// TIA Portal V16 program export: 0 tag tables, 0 data types, 0 data blocks, 4 code blocks (in call order from the OBs), 0 instance data blocks

ORGANIZATION_BLOCK "Main"   // OB1, LAD, ProgramCycle
TITLE = "Main Program Sweep (Cycle)"
{ S7_Optimized_Access := 'TRUE' }
VERSION : 0.1
// stored: AutoNumber true, IsIECCheckEnabled false, SetENOAutomatically false
   VAR_INPUT
      Initial_Call : Bool;   // Initial call of this OB
      Remanence : Bool;   // =True, if remanent data are available
   END_VAR
BEGIN

REGION Network 1
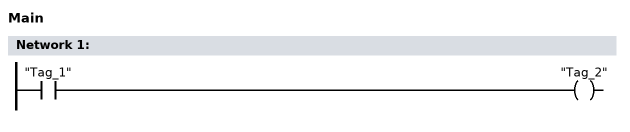
   RUNG wire#powerrail
      Contact( "Tag_1" )
      Coil( "Tag_2" )
   END_RUNG
   // the same network as SCL:
   "Tag_2" := "Tag_1";
END_REGION
END_ORGANIZATION_BLOCK

FUNCTION_BLOCK "FB1_TESTES"   // FB1, LAD
TITLE = FB para lógicas de testes durante start-up
{ S7_Optimized_Access := 'FALSE' }
AUTHOR : AUT_SIST
NAME : RGrn
VERSION : 0.1
// stored: AutoNumber false, IsIECCheckEnabled false, SetENOAutomatically false, UDAEnableTagReadback false
   VAR DB_SPECIFIC
      TESTE : Bool;
      bit_0_1 : Bool;
      bit_0_2 : Bool;
      bit_0_3 : Bool;
      bit_0_4 : Bool;
      bit_0_5 : Bool;
      bit_0_6 : Bool;
      bit_0_7 : Bool;
      bit_1_0 : Bool;
      bit_1_1 : Bool;
      bit_1_2 : Bool;
      bit_1_3 : Bool;
      bit_1_4 : Bool;
      bit_1_5 : Bool;
      bit_1_6 : Bool;
      bit_1_7 : Bool;
      eBosch_FO1_InCy : Bool;
      eBosch_FO1_CyCmp : Bool;
      eBosch_Ch0_1_OK : Bool;
      eBosch_Ch0_2_OK : Bool;
      eBosch_Ch0_3_OK : Bool;
      eBosch_Ch1_1_OK : Bool;
      eBosch_Ch1_2_OK : Bool;
      eBosch_Ch1_3_OK : Bool;
      eBosch_FO2_InCy : Bool;
      eBosch_FO2_CyCmp : Bool;
      eBosch_Ch2_1_OK : Bool;
      eBosch_Ch2_2_OK : Bool;
      eBosch_Ch2_3_OK : Bool;
      eBosch_Ch2_4_OK : Bool;
      bit_3_6 : Bool;
      bit_3_7 : Bool;
      bit_4_0 : Bool;
      bit_4_1 : Bool;
      bit_4_2 : Bool;
      bit_4_3 : Bool;
      bit_4_4 : Bool;
      bit_4_5 : Bool;
      bit_4_6 : Bool;
      bit_4_7 : Bool;
      FP_0 : Bool;
      FP_1 : Bool;
      FP_2 : Bool;
      FP_3 : Bool;
      FP_4 : Bool;
      FP_5 : Bool;
      FP_6 : Bool;
      FP_7 : Bool;
   END_VAR
   VAR_TEMP
      RET_VAL_FC455 : Word;
      Aux_Soma_rodas : Real;
      Med_Rot_rodas : Real;
      Med_parcial_rel_trm : Real;
      Retval_SFC20 : Int;   // Auxiliar armazenamento de mensagens do SFC20
      zero : DWord;
   END_VAR
BEGIN
END_FUNCTION_BLOCK

FUNCTION "FC180_STATUS" : Void   // FC180, LAD
TITLE = Status
{ S7_Optimized_Access := 'TRUE' }
VERSION : 0.1
// stored: AutoNumber false, IsIECCheckEnabled false, SetENOAutomatically false, UDAEnableTagReadback false
   VAR_TEMP
      DB180 : DB_ANY;
   END_VAR
BEGIN

REGION Network 1: DB_ANY CARREGA DB DE REFERENCIA NA VARIAVEL DE INDEXAÇÃO
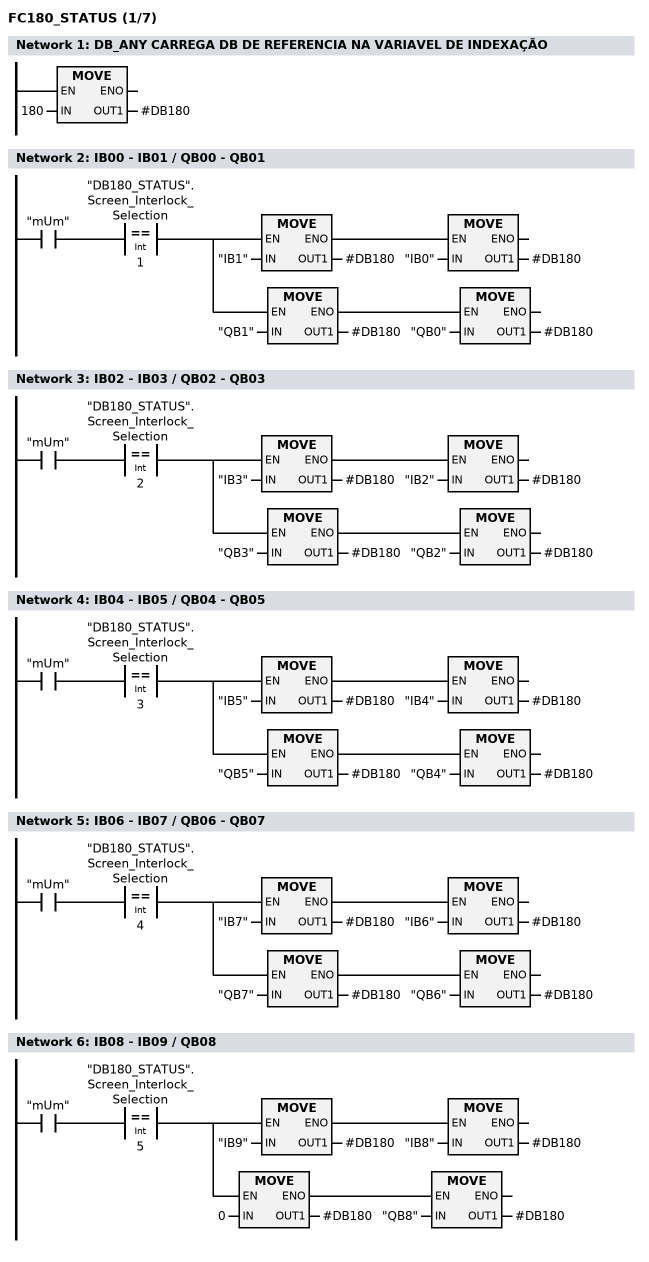
   RUNG wire#powerrail
      Move(in := 180, out1 => #DB180)
   END_RUNG
   // the same network as SCL:
   #DB180 := 180;
END_REGION

REGION Network 2: IB00 - IB01 / QB00 - QB01
   RUNG wire#powerrail
      Contact( "mUm" )
      { S7_Templates := "SrcType := Int" } EQ_Contact(in1 := "DB180_STATUS".Screen_Interlock_Selection, in2 := 1)
      wire#w1
      Move(in := "IB1", out1 => #DB180)
      Move(in := "IB0", out1 => #DB180)
   END_RUNG
   RUNG wire#w1
      Move(in := "QB1", out1 => #DB180)
      Move(in := "QB0", out1 => #DB180)
   END_RUNG
   // the same network as SCL:
   IF "mUm" AND ("DB180_STATUS".Screen_Interlock_Selection = 1) THEN
       #DB180 := "IB1";
       #DB180 := "IB0";
       #DB180 := "QB1";
       #DB180 := "QB0";
   END_IF;
END_REGION

REGION Network 3: IB02 - IB03 / QB02 - QB03
   RUNG wire#powerrail
      Contact( "mUm" )
      { S7_Templates := "SrcType := Int" } EQ_Contact(in1 := "DB180_STATUS".Screen_Interlock_Selection, in2 := 2)
      wire#w1
      Move(in := "IB3", out1 => #DB180)
      Move(in := "IB2", out1 => #DB180)
   END_RUNG
   RUNG wire#w1
      Move(in := "QB3", out1 => #DB180)
      Move(in := "QB2", out1 => #DB180)
   END_RUNG
   // the same network as SCL:
   IF "mUm" AND ("DB180_STATUS".Screen_Interlock_Selection = 2) THEN
       #DB180 := "IB3";
       #DB180 := "IB2";
       #DB180 := "QB3";
       #DB180 := "QB2";
   END_IF;
END_REGION

REGION Network 4: IB04 - IB05 / QB04 - QB05
   RUNG wire#powerrail
      Contact( "mUm" )
      { S7_Templates := "SrcType := Int" } EQ_Contact(in1 := "DB180_STATUS".Screen_Interlock_Selection, in2 := 3)
      wire#w1
      Move(in := "IB5", out1 => #DB180)
      Move(in := "IB4", out1 => #DB180)
   END_RUNG
   RUNG wire#w1
      Move(in := "QB5", out1 => #DB180)
      Move(in := "QB4", out1 => #DB180)
   END_RUNG
   // the same network as SCL:
   IF "mUm" AND ("DB180_STATUS".Screen_Interlock_Selection = 3) THEN
       #DB180 := "IB5";
       #DB180 := "IB4";
       #DB180 := "QB5";
       #DB180 := "QB4";
   END_IF;
END_REGION

REGION Network 5: IB06 - IB07 / QB06 - QB07
   RUNG wire#powerrail
      Contact( "mUm" )
      { S7_Templates := "SrcType := Int" } EQ_Contact(in1 := "DB180_STATUS".Screen_Interlock_Selection, in2 := 4)
      wire#w1
      Move(in := "IB7", out1 => #DB180)
      Move(in := "IB6", out1 => #DB180)
   END_RUNG
   RUNG wire#w1
      Move(in := "QB7", out1 => #DB180)
      Move(in := "QB6", out1 => #DB180)
   END_RUNG
   // the same network as SCL:
   IF "mUm" AND ("DB180_STATUS".Screen_Interlock_Selection = 4) THEN
       #DB180 := "IB7";
       #DB180 := "IB6";
       #DB180 := "QB7";
       #DB180 := "QB6";
   END_IF;
END_REGION

REGION Network 6: IB08 - IB09 / QB08
   RUNG wire#powerrail
      Contact( "mUm" )
      { S7_Templates := "SrcType := Int" } EQ_Contact(in1 := "DB180_STATUS".Screen_Interlock_Selection, in2 := 5)
      wire#w1
      Move(in := "IB9", out1 => #DB180)
      Move(in := "IB8", out1 => #DB180)
   END_RUNG
   RUNG wire#w1
      Move(in := 0, out1 => #DB180)
      Move(in := "QB8", out1 => #DB180)
   END_RUNG
   // the same network as SCL:
   IF "mUm" AND ("DB180_STATUS".Screen_Interlock_Selection = 5) THEN
       #DB180 := "IB9";
       #DB180 := "IB8";
       #DB180 := 0;
       #DB180 := "QB8";
   END_IF;
END_REGION

REGION Network 7: IB21 - IB23 / QB20 - QB22
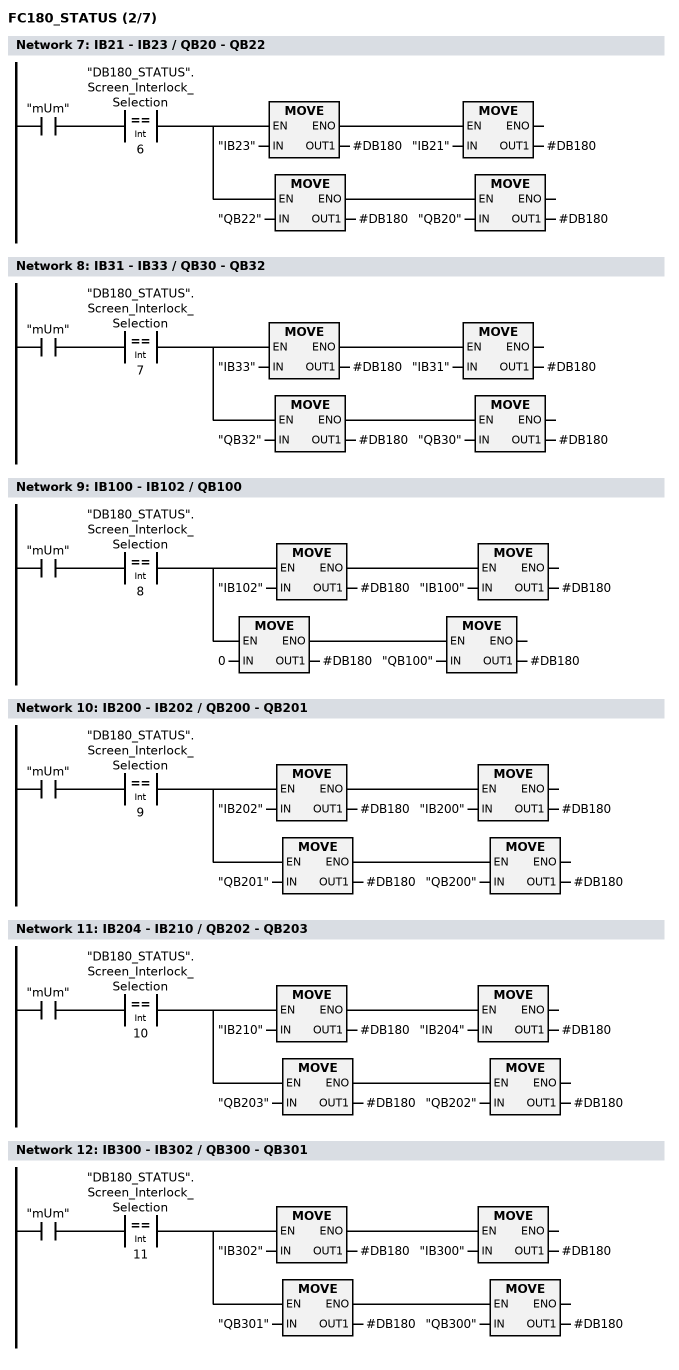
   RUNG wire#powerrail
      Contact( "mUm" )
      { S7_Templates := "SrcType := Int" } EQ_Contact(in1 := "DB180_STATUS".Screen_Interlock_Selection, in2 := 6)
      wire#w1
      Move(in := "IB23", out1 => #DB180)
      Move(in := "IB21", out1 => #DB180)
   END_RUNG
   RUNG wire#w1
      Move(in := "QB22", out1 => #DB180)
      Move(in := "QB20", out1 => #DB180)
   END_RUNG
   // the same network as SCL:
   IF "mUm" AND ("DB180_STATUS".Screen_Interlock_Selection = 6) THEN
       #DB180 := "IB23";
       #DB180 := "IB21";
       #DB180 := "QB22";
       #DB180 := "QB20";
   END_IF;
END_REGION

REGION Network 8: IB31 - IB33 / QB30 - QB32
   RUNG wire#powerrail
      Contact( "mUm" )
      { S7_Templates := "SrcType := Int" } EQ_Contact(in1 := "DB180_STATUS".Screen_Interlock_Selection, in2 := 7)
      wire#w1
      Move(in := "IB33", out1 => #DB180)
      Move(in := "IB31", out1 => #DB180)
   END_RUNG
   RUNG wire#w1
      Move(in := "QB32", out1 => #DB180)
      Move(in := "QB30", out1 => #DB180)
   END_RUNG
   // the same network as SCL:
   IF "mUm" AND ("DB180_STATUS".Screen_Interlock_Selection = 7) THEN
       #DB180 := "IB33";
       #DB180 := "IB31";
       #DB180 := "QB32";
       #DB180 := "QB30";
   END_IF;
END_REGION

REGION Network 9: IB100 - IB102 / QB100
   RUNG wire#powerrail
      Contact( "mUm" )
      { S7_Templates := "SrcType := Int" } EQ_Contact(in1 := "DB180_STATUS".Screen_Interlock_Selection, in2 := 8)
      wire#w1
      Move(in := "IB102", out1 => #DB180)
      Move(in := "IB100", out1 => #DB180)
   END_RUNG
   RUNG wire#w1
      Move(in := 0, out1 => #DB180)
      Move(in := "QB100", out1 => #DB180)
   END_RUNG
   // the same network as SCL:
   IF "mUm" AND ("DB180_STATUS".Screen_Interlock_Selection = 8) THEN
       #DB180 := "IB102";
       #DB180 := "IB100";
       #DB180 := 0;
       #DB180 := "QB100";
   END_IF;
END_REGION

REGION Network 10: IB200 - IB202 / QB200 - QB201
   RUNG wire#powerrail
      Contact( "mUm" )
      { S7_Templates := "SrcType := Int" } EQ_Contact(in1 := "DB180_STATUS".Screen_Interlock_Selection, in2 := 9)
      wire#w1
      Move(in := "IB202", out1 => #DB180)
      Move(in := "IB200", out1 => #DB180)
   END_RUNG
   RUNG wire#w1
      Move(in := "QB201", out1 => #DB180)
      Move(in := "QB200", out1 => #DB180)
   END_RUNG
   // the same network as SCL:
   IF "mUm" AND ("DB180_STATUS".Screen_Interlock_Selection = 9) THEN
       #DB180 := "IB202";
       #DB180 := "IB200";
       #DB180 := "QB201";
       #DB180 := "QB200";
   END_IF;
END_REGION

REGION Network 11: IB204 - IB210 / QB202 - QB203
   RUNG wire#powerrail
      Contact( "mUm" )
      { S7_Templates := "SrcType := Int" } EQ_Contact(in1 := "DB180_STATUS".Screen_Interlock_Selection, in2 := 10)
      wire#w1
      Move(in := "IB210", out1 => #DB180)
      Move(in := "IB204", out1 => #DB180)
   END_RUNG
   RUNG wire#w1
      Move(in := "QB203", out1 => #DB180)
      Move(in := "QB202", out1 => #DB180)
   END_RUNG
   // the same network as SCL:
   IF "mUm" AND ("DB180_STATUS".Screen_Interlock_Selection = 10) THEN
       #DB180 := "IB210";
       #DB180 := "IB204";
       #DB180 := "QB203";
       #DB180 := "QB202";
   END_IF;
END_REGION

REGION Network 12: IB300 - IB302 / QB300 - QB301
   RUNG wire#powerrail
      Contact( "mUm" )
      { S7_Templates := "SrcType := Int" } EQ_Contact(in1 := "DB180_STATUS".Screen_Interlock_Selection, in2 := 11)
      wire#w1
      Move(in := "IB302", out1 => #DB180)
      Move(in := "IB300", out1 => #DB180)
   END_RUNG
   RUNG wire#w1
      Move(in := "QB301", out1 => #DB180)
      Move(in := "QB300", out1 => #DB180)
   END_RUNG
   // the same network as SCL:
   IF "mUm" AND ("DB180_STATUS".Screen_Interlock_Selection = 11) THEN
       #DB180 := "IB302";
       #DB180 := "IB300";
       #DB180 := "QB301";
       #DB180 := "QB300";
   END_IF;
END_REGION

REGION Network 13: IB304 - IB306 / QB302 - QB303
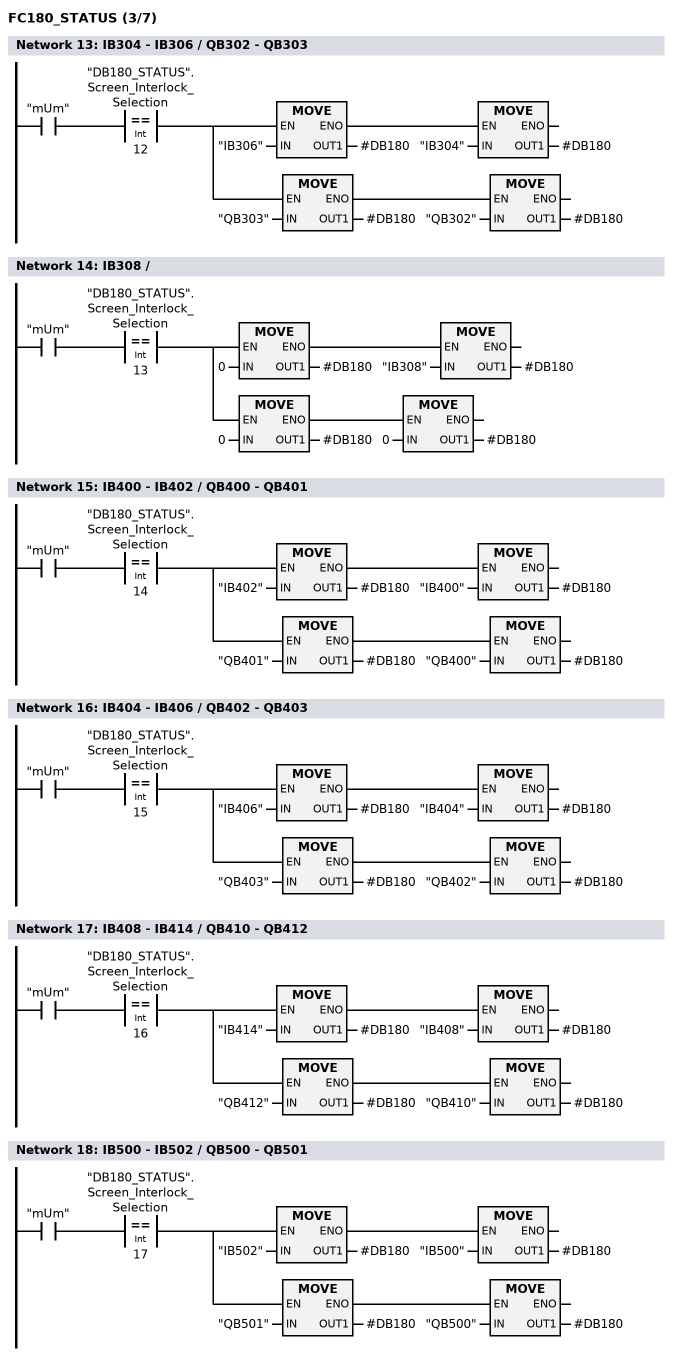
   RUNG wire#powerrail
      Contact( "mUm" )
      { S7_Templates := "SrcType := Int" } EQ_Contact(in1 := "DB180_STATUS".Screen_Interlock_Selection, in2 := 12)
      wire#w1
      Move(in := "IB306", out1 => #DB180)
      Move(in := "IB304", out1 => #DB180)
   END_RUNG
   RUNG wire#w1
      Move(in := "QB303", out1 => #DB180)
      Move(in := "QB302", out1 => #DB180)
   END_RUNG
   // the same network as SCL:
   IF "mUm" AND ("DB180_STATUS".Screen_Interlock_Selection = 12) THEN
       #DB180 := "IB306";
       #DB180 := "IB304";
       #DB180 := "QB303";
       #DB180 := "QB302";
   END_IF;
END_REGION

REGION Network 14: IB308 /
   RUNG wire#powerrail
      Contact( "mUm" )
      { S7_Templates := "SrcType := Int" } EQ_Contact(in1 := "DB180_STATUS".Screen_Interlock_Selection, in2 := 13)
      wire#w1
      Move(in := 0, out1 => #DB180)
      Move(in := "IB308", out1 => #DB180)
   END_RUNG
   RUNG wire#w1
      Move(in := 0, out1 => #DB180)
      Move(in := 0, out1 => #DB180)
   END_RUNG
   // the same network as SCL:
   IF "mUm" AND ("DB180_STATUS".Screen_Interlock_Selection = 13) THEN
       #DB180 := 0;
       #DB180 := "IB308";
       #DB180 := 0;
       #DB180 := 0;
   END_IF;
END_REGION

REGION Network 15: IB400 - IB402 / QB400 - QB401
   RUNG wire#powerrail
      Contact( "mUm" )
      { S7_Templates := "SrcType := Int" } EQ_Contact(in1 := "DB180_STATUS".Screen_Interlock_Selection, in2 := 14)
      wire#w1
      Move(in := "IB402", out1 => #DB180)
      Move(in := "IB400", out1 => #DB180)
   END_RUNG
   RUNG wire#w1
      Move(in := "QB401", out1 => #DB180)
      Move(in := "QB400", out1 => #DB180)
   END_RUNG
   // the same network as SCL:
   IF "mUm" AND ("DB180_STATUS".Screen_Interlock_Selection = 14) THEN
       #DB180 := "IB402";
       #DB180 := "IB400";
       #DB180 := "QB401";
       #DB180 := "QB400";
   END_IF;
END_REGION

REGION Network 16: IB404 - IB406 / QB402 - QB403
   RUNG wire#powerrail
      Contact( "mUm" )
      { S7_Templates := "SrcType := Int" } EQ_Contact(in1 := "DB180_STATUS".Screen_Interlock_Selection, in2 := 15)
      wire#w1
      Move(in := "IB406", out1 => #DB180)
      Move(in := "IB404", out1 => #DB180)
   END_RUNG
   RUNG wire#w1
      Move(in := "QB403", out1 => #DB180)
      Move(in := "QB402", out1 => #DB180)
   END_RUNG
   // the same network as SCL:
   IF "mUm" AND ("DB180_STATUS".Screen_Interlock_Selection = 15) THEN
       #DB180 := "IB406";
       #DB180 := "IB404";
       #DB180 := "QB403";
       #DB180 := "QB402";
   END_IF;
END_REGION

REGION Network 17: IB408 - IB414 / QB410 - QB412
   RUNG wire#powerrail
      Contact( "mUm" )
      { S7_Templates := "SrcType := Int" } EQ_Contact(in1 := "DB180_STATUS".Screen_Interlock_Selection, in2 := 16)
      wire#w1
      Move(in := "IB414", out1 => #DB180)
      Move(in := "IB408", out1 => #DB180)
   END_RUNG
   RUNG wire#w1
      Move(in := "QB412", out1 => #DB180)
      Move(in := "QB410", out1 => #DB180)
   END_RUNG
   // the same network as SCL:
   IF "mUm" AND ("DB180_STATUS".Screen_Interlock_Selection = 16) THEN
       #DB180 := "IB414";
       #DB180 := "IB408";
       #DB180 := "QB412";
       #DB180 := "QB410";
   END_IF;
END_REGION

REGION Network 18: IB500 - IB502 / QB500 - QB501
   RUNG wire#powerrail
      Contact( "mUm" )
      { S7_Templates := "SrcType := Int" } EQ_Contact(in1 := "DB180_STATUS".Screen_Interlock_Selection, in2 := 17)
      wire#w1
      Move(in := "IB502", out1 => #DB180)
      Move(in := "IB500", out1 => #DB180)
   END_RUNG
   RUNG wire#w1
      Move(in := "QB501", out1 => #DB180)
      Move(in := "QB500", out1 => #DB180)
   END_RUNG
   // the same network as SCL:
   IF "mUm" AND ("DB180_STATUS".Screen_Interlock_Selection = 17) THEN
       #DB180 := "IB502";
       #DB180 := "IB500";
       #DB180 := "QB501";
       #DB180 := "QB500";
   END_IF;
END_REGION

REGION Network 19: IB504 - IB506 / QB502 - QB503
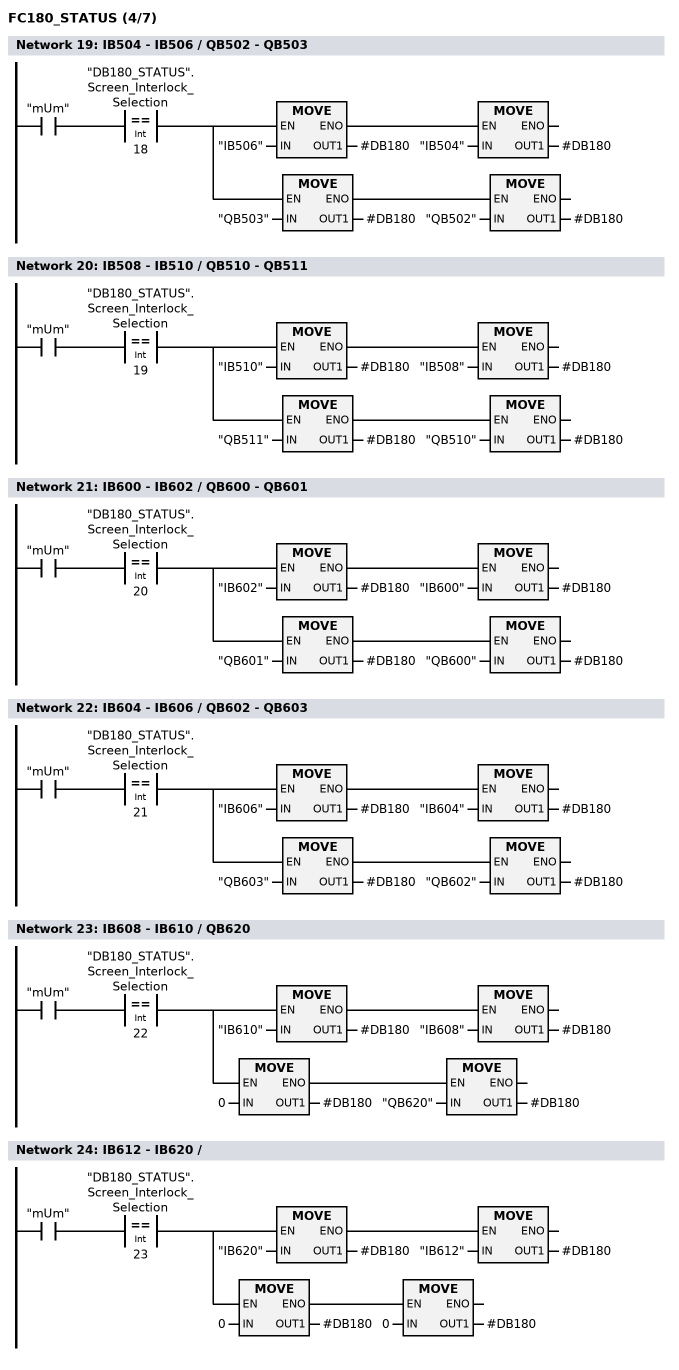
   RUNG wire#powerrail
      Contact( "mUm" )
      { S7_Templates := "SrcType := Int" } EQ_Contact(in1 := "DB180_STATUS".Screen_Interlock_Selection, in2 := 18)
      wire#w1
      Move(in := "IB506", out1 => #DB180)
      Move(in := "IB504", out1 => #DB180)
   END_RUNG
   RUNG wire#w1
      Move(in := "QB503", out1 => #DB180)
      Move(in := "QB502", out1 => #DB180)
   END_RUNG
   // the same network as SCL:
   IF "mUm" AND ("DB180_STATUS".Screen_Interlock_Selection = 18) THEN
       #DB180 := "IB506";
       #DB180 := "IB504";
       #DB180 := "QB503";
       #DB180 := "QB502";
   END_IF;
END_REGION

REGION Network 20: IB508 - IB510 / QB510 - QB511
   RUNG wire#powerrail
      Contact( "mUm" )
      { S7_Templates := "SrcType := Int" } EQ_Contact(in1 := "DB180_STATUS".Screen_Interlock_Selection, in2 := 19)
      wire#w1
      Move(in := "IB510", out1 => #DB180)
      Move(in := "IB508", out1 => #DB180)
   END_RUNG
   RUNG wire#w1
      Move(in := "QB511", out1 => #DB180)
      Move(in := "QB510", out1 => #DB180)
   END_RUNG
   // the same network as SCL:
   IF "mUm" AND ("DB180_STATUS".Screen_Interlock_Selection = 19) THEN
       #DB180 := "IB510";
       #DB180 := "IB508";
       #DB180 := "QB511";
       #DB180 := "QB510";
   END_IF;
END_REGION

REGION Network 21: IB600 - IB602 / QB600 - QB601
   RUNG wire#powerrail
      Contact( "mUm" )
      { S7_Templates := "SrcType := Int" } EQ_Contact(in1 := "DB180_STATUS".Screen_Interlock_Selection, in2 := 20)
      wire#w1
      Move(in := "IB602", out1 => #DB180)
      Move(in := "IB600", out1 => #DB180)
   END_RUNG
   RUNG wire#w1
      Move(in := "QB601", out1 => #DB180)
      Move(in := "QB600", out1 => #DB180)
   END_RUNG
   // the same network as SCL:
   IF "mUm" AND ("DB180_STATUS".Screen_Interlock_Selection = 20) THEN
       #DB180 := "IB602";
       #DB180 := "IB600";
       #DB180 := "QB601";
       #DB180 := "QB600";
   END_IF;
END_REGION

REGION Network 22: IB604 - IB606 / QB602 - QB603
   RUNG wire#powerrail
      Contact( "mUm" )
      { S7_Templates := "SrcType := Int" } EQ_Contact(in1 := "DB180_STATUS".Screen_Interlock_Selection, in2 := 21)
      wire#w1
      Move(in := "IB606", out1 => #DB180)
      Move(in := "IB604", out1 => #DB180)
   END_RUNG
   RUNG wire#w1
      Move(in := "QB603", out1 => #DB180)
      Move(in := "QB602", out1 => #DB180)
   END_RUNG
   // the same network as SCL:
   IF "mUm" AND ("DB180_STATUS".Screen_Interlock_Selection = 21) THEN
       #DB180 := "IB606";
       #DB180 := "IB604";
       #DB180 := "QB603";
       #DB180 := "QB602";
   END_IF;
END_REGION

REGION Network 23: IB608 - IB610 / QB620
   RUNG wire#powerrail
      Contact( "mUm" )
      { S7_Templates := "SrcType := Int" } EQ_Contact(in1 := "DB180_STATUS".Screen_Interlock_Selection, in2 := 22)
      wire#w1
      Move(in := "IB610", out1 => #DB180)
      Move(in := "IB608", out1 => #DB180)
   END_RUNG
   RUNG wire#w1
      Move(in := 0, out1 => #DB180)
      Move(in := "QB620", out1 => #DB180)
   END_RUNG
   // the same network as SCL:
   IF "mUm" AND ("DB180_STATUS".Screen_Interlock_Selection = 22) THEN
       #DB180 := "IB610";
       #DB180 := "IB608";
       #DB180 := 0;
       #DB180 := "QB620";
   END_IF;
END_REGION

REGION Network 24: IB612 - IB620 /
   RUNG wire#powerrail
      Contact( "mUm" )
      { S7_Templates := "SrcType := Int" } EQ_Contact(in1 := "DB180_STATUS".Screen_Interlock_Selection, in2 := 23)
      wire#w1
      Move(in := "IB620", out1 => #DB180)
      Move(in := "IB612", out1 => #DB180)
   END_RUNG
   RUNG wire#w1
      Move(in := 0, out1 => #DB180)
      Move(in := 0, out1 => #DB180)
   END_RUNG
   // the same network as SCL:
   IF "mUm" AND ("DB180_STATUS".Screen_Interlock_Selection = 23) THEN
       #DB180 := "IB620";
       #DB180 := "IB612";
       #DB180 := 0;
       #DB180 := 0;
   END_IF;
END_REGION

REGION Network 25: IB700 /
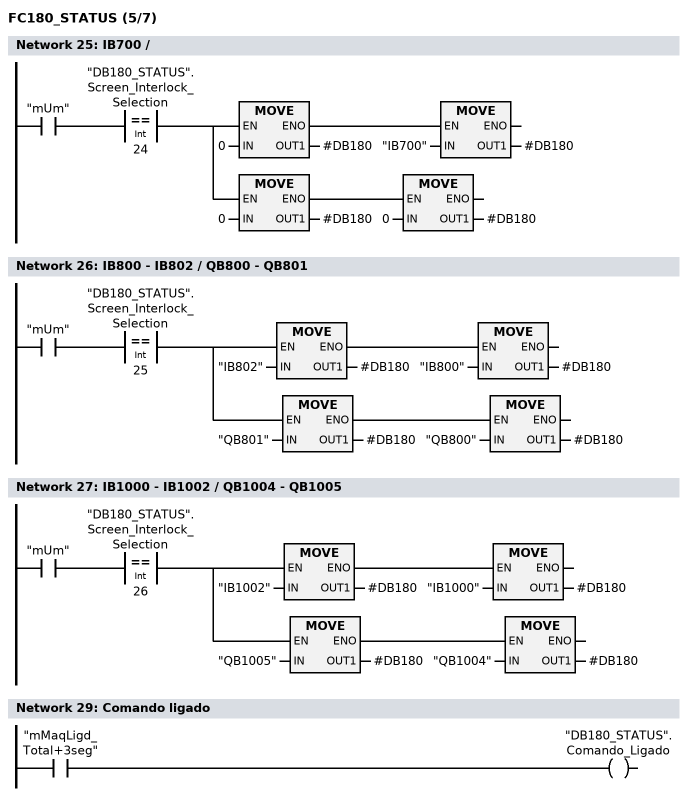
   RUNG wire#powerrail
      Contact( "mUm" )
      { S7_Templates := "SrcType := Int" } EQ_Contact(in1 := "DB180_STATUS".Screen_Interlock_Selection, in2 := 24)
      wire#w1
      Move(in := 0, out1 => #DB180)
      Move(in := "IB700", out1 => #DB180)
   END_RUNG
   RUNG wire#w1
      Move(in := 0, out1 => #DB180)
      Move(in := 0, out1 => #DB180)
   END_RUNG
   // the same network as SCL:
   IF "mUm" AND ("DB180_STATUS".Screen_Interlock_Selection = 24) THEN
       #DB180 := 0;
       #DB180 := "IB700";
       #DB180 := 0;
       #DB180 := 0;
   END_IF;
END_REGION

REGION Network 26: IB800 - IB802 / QB800 - QB801
   RUNG wire#powerrail
      Contact( "mUm" )
      { S7_Templates := "SrcType := Int" } EQ_Contact(in1 := "DB180_STATUS".Screen_Interlock_Selection, in2 := 25)
      wire#w1
      Move(in := "IB802", out1 => #DB180)
      Move(in := "IB800", out1 => #DB180)
   END_RUNG
   RUNG wire#w1
      Move(in := "QB801", out1 => #DB180)
      Move(in := "QB800", out1 => #DB180)
   END_RUNG
   // the same network as SCL:
   IF "mUm" AND ("DB180_STATUS".Screen_Interlock_Selection = 25) THEN
       #DB180 := "IB802";
       #DB180 := "IB800";
       #DB180 := "QB801";
       #DB180 := "QB800";
   END_IF;
END_REGION

REGION Network 27: IB1000 - IB1002 / QB1004 - QB1005
   RUNG wire#powerrail
      Contact( "mUm" )
      { S7_Templates := "SrcType := Int" } EQ_Contact(in1 := "DB180_STATUS".Screen_Interlock_Selection, in2 := 26)
      wire#w1
      Move(in := "IB1002", out1 => #DB180)
      Move(in := "IB1000", out1 => #DB180)
   END_RUNG
   RUNG wire#w1
      Move(in := "QB1005", out1 => #DB180)
      Move(in := "QB1004", out1 => #DB180)
   END_RUNG
   // the same network as SCL:
   IF "mUm" AND ("DB180_STATUS".Screen_Interlock_Selection = 26) THEN
       #DB180 := "IB1002";
       #DB180 := "IB1000";
       #DB180 := "QB1005";
       #DB180 := "QB1004";
   END_IF;
END_REGION

REGION Network 28: Status Comando
END_REGION

REGION Network 29: Comando ligado
   RUNG wire#powerrail
      Contact( "mMaqLigd_Total+3seg" )
      Coil( "DB180_STATUS".Comando_Ligado )
   END_RUNG
   // the same network as SCL:
   "DB180_STATUS".Comando_Ligado := "mMaqLigd_Total+3seg";
END_REGION

REGION Network 30: Alarme Presente
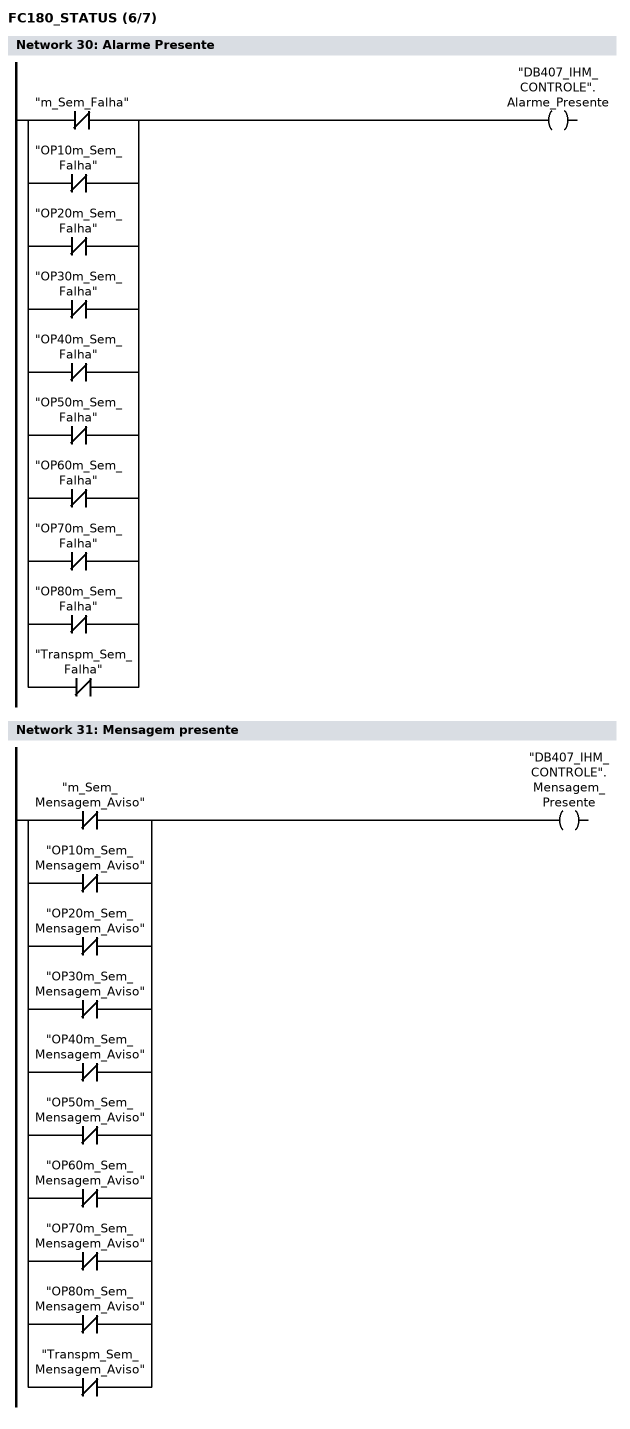
   RUNG wire#powerrail
      I_Contact( "m_Sem_Falha" )
      wire#w1
      Coil( "DB407_IHM_CONTROLE".Alarme_Presente )
   END_RUNG
   RUNG wire#powerrail
      I_Contact( "OP10m_Sem_Falha" )
   END_RUNG wire#w1
   RUNG wire#powerrail
      I_Contact( "OP20m_Sem_Falha" )
   END_RUNG wire#w1
   RUNG wire#powerrail
      I_Contact( "OP30m_Sem_Falha" )
   END_RUNG wire#w1
   RUNG wire#powerrail
      I_Contact( "OP40m_Sem_Falha" )
   END_RUNG wire#w1
   RUNG wire#powerrail
      I_Contact( "OP50m_Sem_Falha" )
   END_RUNG wire#w1
   RUNG wire#powerrail
      I_Contact( "OP60m_Sem_Falha" )
   END_RUNG wire#w1
   RUNG wire#powerrail
      I_Contact( "OP70m_Sem_Falha" )
   END_RUNG wire#w1
   RUNG wire#powerrail
      I_Contact( "OP80m_Sem_Falha" )
   END_RUNG wire#w1
   RUNG wire#powerrail
      I_Contact( "Transpm_Sem_Falha" )
   END_RUNG wire#w1
   // the same network as SCL:
   "DB407_IHM_CONTROLE".Alarme_Presente := NOT "m_Sem_Falha" OR NOT "OP10m_Sem_Falha" OR NOT "OP20m_Sem_Falha" OR NOT "OP30m_Sem_Falha" OR NOT "OP40m_Sem_Falha" OR NOT "OP50m_Sem_Falha" OR NOT "OP60m_Sem_Falha" OR NOT "OP70m_Sem_Falha" OR NOT "OP80m_Sem_Falha" OR NOT "Transpm_Sem_Falha";
END_REGION

REGION Network 31: Mensagem presente
   RUNG wire#powerrail
      I_Contact( "m_Sem_Mensagem_Aviso" )
      wire#w1
      Coil( "DB407_IHM_CONTROLE".Mensagem_Presente )
   END_RUNG
   RUNG wire#powerrail
      I_Contact( "OP10m_Sem_Mensagem_Aviso" )
   END_RUNG wire#w1
   RUNG wire#powerrail
      I_Contact( "OP20m_Sem_Mensagem_Aviso" )
   END_RUNG wire#w1
   RUNG wire#powerrail
      I_Contact( "OP30m_Sem_Mensagem_Aviso" )
   END_RUNG wire#w1
   RUNG wire#powerrail
      I_Contact( "OP40m_Sem_Mensagem_Aviso" )
   END_RUNG wire#w1
   RUNG wire#powerrail
      I_Contact( "OP50m_Sem_Mensagem_Aviso" )
   END_RUNG wire#w1
   RUNG wire#powerrail
      I_Contact( "OP60m_Sem_Mensagem_Aviso" )
   END_RUNG wire#w1
   RUNG wire#powerrail
      I_Contact( "OP70m_Sem_Mensagem_Aviso" )
   END_RUNG wire#w1
   RUNG wire#powerrail
      I_Contact( "OP80m_Sem_Mensagem_Aviso" )
   END_RUNG wire#w1
   RUNG wire#powerrail
      I_Contact( "Transpm_Sem_Mensagem_Aviso" )
   END_RUNG wire#w1
   // the same network as SCL:
   "DB407_IHM_CONTROLE".Mensagem_Presente := NOT "m_Sem_Mensagem_Aviso" OR NOT "OP10m_Sem_Mensagem_Aviso" OR NOT "OP20m_Sem_Mensagem_Aviso" OR NOT "OP30m_Sem_Mensagem_Aviso" OR NOT "OP40m_Sem_Mensagem_Aviso" OR NOT "OP50m_Sem_Mensagem_Aviso" OR NOT "OP60m_Sem_Mensagem_Aviso" OR NOT "OP70m_Sem_Mensagem_Aviso" OR NOT "OP80m_Sem_Mensagem_Aviso" OR NOT "Transpm_Sem_Mensagem_Aviso";
END_REGION

REGION Network 32: Bloqueio Presente
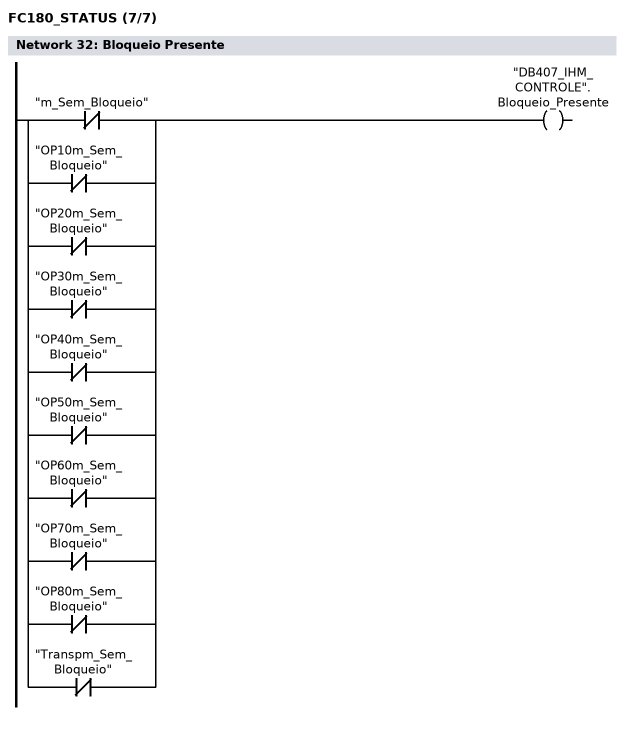
   RUNG wire#powerrail
      I_Contact( "m_Sem_Bloqueio" )
      wire#w1
      Coil( "DB407_IHM_CONTROLE".Bloqueio_Presente )
   END_RUNG
   RUNG wire#powerrail
      I_Contact( "OP10m_Sem_Bloqueio" )
   END_RUNG wire#w1
   RUNG wire#powerrail
      I_Contact( "OP20m_Sem_Bloqueio" )
   END_RUNG wire#w1
   RUNG wire#powerrail
      I_Contact( "OP30m_Sem_Bloqueio" )
   END_RUNG wire#w1
   RUNG wire#powerrail
      I_Contact( "OP40m_Sem_Bloqueio" )
   END_RUNG wire#w1
   RUNG wire#powerrail
      I_Contact( "OP50m_Sem_Bloqueio" )
   END_RUNG wire#w1
   RUNG wire#powerrail
      I_Contact( "OP60m_Sem_Bloqueio" )
   END_RUNG wire#w1
   RUNG wire#powerrail
      I_Contact( "OP70m_Sem_Bloqueio" )
   END_RUNG wire#w1
   RUNG wire#powerrail
      I_Contact( "OP80m_Sem_Bloqueio" )
   END_RUNG wire#w1
   RUNG wire#powerrail
      I_Contact( "Transpm_Sem_Bloqueio" )
   END_RUNG wire#w1
   // the same network as SCL:
   "DB407_IHM_CONTROLE".Bloqueio_Presente := NOT "m_Sem_Bloqueio" OR NOT "OP10m_Sem_Bloqueio" OR NOT "OP20m_Sem_Bloqueio" OR NOT "OP30m_Sem_Bloqueio" OR NOT "OP40m_Sem_Bloqueio" OR NOT "OP50m_Sem_Bloqueio" OR NOT "OP60m_Sem_Bloqueio" OR NOT "OP70m_Sem_Bloqueio" OR NOT "OP80m_Sem_Bloqueio" OR NOT "Transpm_Sem_Bloqueio";
END_REGION
END_FUNCTION

FUNCTION "MainFC" : Void   // FC1, LAD
{ S7_Optimized_Access := 'TRUE' }
VERSION : 0.1
// stored: AutoNumber true, IsIECCheckEnabled false, SetENOAutomatically false, UDAEnableTagReadback false
BEGIN

REGION Network 1
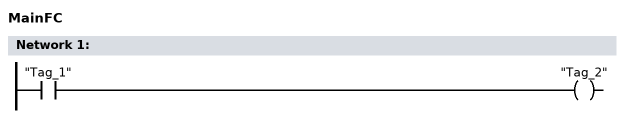
   RUNG wire#powerrail
      Contact( "Tag_1" )
      Coil( "Tag_2" )
   END_RUNG
   // the same network as SCL:
   "Tag_2" := "Tag_1";
END_REGION
END_FUNCTION
